FUNCTION_BLOCK "FB_Frequency_Inverter"   // FB6, LAD
{ S7_Optimized_Access := 'TRUE' }
// stored: AutoNumber false, MemoryReserve 100, SetENOAutomatically false
   VAR_INPUT
      Emergency_Stop_Release : Bool;
      Start : Bool;
      Manual_Turn_On_Motor : Bool;
      Pause_Conveyor_Belt_And_Carousel_Functional_Test : Bool;
      Select_Motor_Speedy : SInt;
   END_VAR
   VAR_OUTPUT
      Motor_Spining_Speedy_1 : Bool;
      Motor_Spining_Speedy_2 : Bool;
      Motor_Spining_Speedy_3 : Bool;
   END_VAR
BEGIN

REGION Network 1
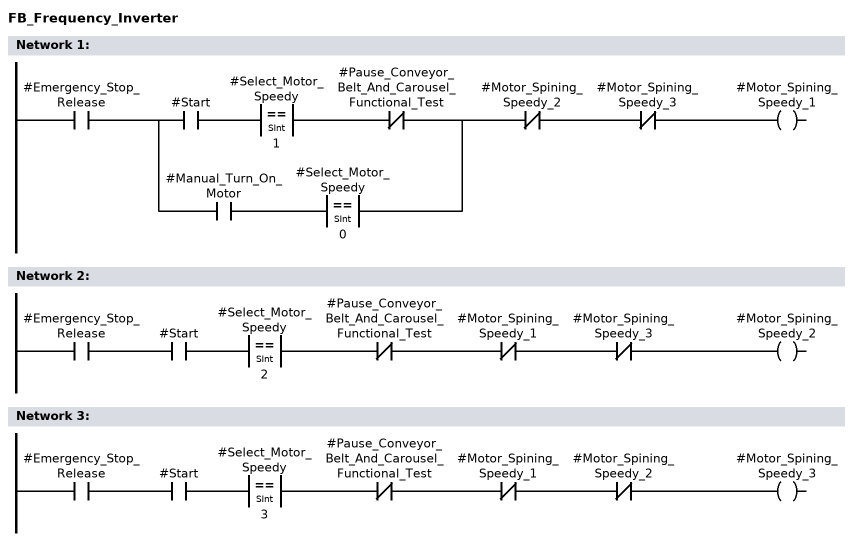
   RUNG wire#powerrail
      Contact( #Emergency_Stop_Release )
      wire#w1
      Contact( #Start )
      { S7_Templates := "SrcType := SInt" } EQ_Contact(in1 := #Select_Motor_Speedy, in2 := 1)
      I_Contact( #Pause_Conveyor_Belt_And_Carousel_Functional_Test )
      wire#w2
      I_Contact( #Motor_Spining_Speedy_2 )
      I_Contact( #Motor_Spining_Speedy_3 )
      Coil( #Motor_Spining_Speedy_1 )
   END_RUNG
   RUNG wire#w1
      Contact( #Manual_Turn_On_Motor )
      { S7_Templates := "SrcType := SInt" } EQ_Contact(in1 := #Select_Motor_Speedy, in2 := 0)
   END_RUNG wire#w2
   // the same network as SCL:
   #Motor_Spining_Speedy_1 := #Emergency_Stop_Release AND ((#Start AND (#Select_Motor_Speedy = 1) AND NOT #Pause_Conveyor_Belt_And_Carousel_Functional_Test) OR (#Manual_Turn_On_Motor AND (#Select_Motor_Speedy = 0))) AND NOT #Motor_Spining_Speedy_2 AND NOT #Motor_Spining_Speedy_3;
END_REGION

REGION Network 2
   RUNG wire#powerrail
      Contact( #Emergency_Stop_Release )
      Contact( #Start )
      { S7_Templates := "SrcType := SInt" } EQ_Contact(in1 := #Select_Motor_Speedy, in2 := 2)
      I_Contact( #Pause_Conveyor_Belt_And_Carousel_Functional_Test )
      I_Contact( #Motor_Spining_Speedy_1 )
      I_Contact( #Motor_Spining_Speedy_3 )
      Coil( #Motor_Spining_Speedy_2 )
   END_RUNG
   // the same network as SCL:
   #Motor_Spining_Speedy_2 := #Emergency_Stop_Release AND #Start AND (#Select_Motor_Speedy = 2) AND NOT #Pause_Conveyor_Belt_And_Carousel_Functional_Test AND NOT #Motor_Spining_Speedy_1 AND NOT #Motor_Spining_Speedy_3;
END_REGION

REGION Network 3
   RUNG wire#powerrail
      Contact( #Emergency_Stop_Release )
      Contact( #Start )
      { S7_Templates := "SrcType := SInt" } EQ_Contact(in1 := #Select_Motor_Speedy, in2 := 3)
      I_Contact( #Pause_Conveyor_Belt_And_Carousel_Functional_Test )
      I_Contact( #Motor_Spining_Speedy_1 )
      I_Contact( #Motor_Spining_Speedy_2 )
      Coil( #Motor_Spining_Speedy_3 )
   END_RUNG
   // the same network as SCL:
   #Motor_Spining_Speedy_3 := #Emergency_Stop_Release AND #Start AND (#Select_Motor_Speedy = 3) AND NOT #Pause_Conveyor_Belt_And_Carousel_Functional_Test AND NOT #Motor_Spining_Speedy_1 AND NOT #Motor_Spining_Speedy_2;
END_REGION
END_FUNCTION_BLOCK

FUNCTION_BLOCK "FB_Send_Water_Fountain_To_Rework"   // FB7, LAD
{ S7_Optimized_Access := 'TRUE' }
// stored: AutoNumber false, MemoryReserve 100, SetENOAutomatically false
   VAR_INPUT
      Emergency_Stop_Release : Bool;
      Start : Bool;
      Water_Fountain_Fail_Test : Bool;
      Trigger_Read_Serial_Number_Exit_Functional_Test : Bool;
      Sensor_Water_Fountain_Exit_Functional_Test_Spinner_Conveyor_Belt : Bool;
      Sensor_Spinner_Exit_Functional_Test_Position_Withdrawn : Bool;
      Sensor_Spinner_Exit_Functional_Test_Position_Advanced : Bool;
      Sensor_Water_Fountain_Exit_Functional_Test_After_Spinner_Conveyor_Belt : Bool;
      Sensor_Water_Fountain_Geting_Entrace_Rework_Conveyor_Belt_Start : Bool;
   END_VAR
   VAR_OUTPUT
      Turn_On_Conveyor_Belt_Motor_Spinner_Get_Exit_Functional_Test : Bool;
      Valve_Advance_Spinner_Get_Exit_Functional_Test : Bool;
      Pause_Conveyor_Belt_And_Carousel_Functional_Test : Bool;
   END_VAR
   VAR
      Aux_Trig_0 : Bool;
      Aux_Trig_1 : Bool;
      Aux_Trig_2 : Bool;
      Aux_Trig_3 : Bool;
      Aux_Trig_4 : Bool;
      Aux_Trig_5 : Bool;
      Aux_Trig_6 : Bool;
      Aux_Trig_7 : Bool;
      Wait_Clean_Spinner : Bool;
      Wait_Get_In_Spinner : Bool;
      "Counter" : USInt;
      Timer_Delay_Turn_On_Motor_Spinner_Conveyor_Belt { S7_SetPoint := 'True'} : TON_TIME;
   END_VAR
   VAR RETAIN
      Counter_Water_Fountain_Exiting_Functional_Test { S7_SetPoint := 'True'} : CTUD_USINT;
   END_VAR
   VAR_TEMP   // added for the SCL form of the ladder/FBD networks
      _w1 : Bool;
      _w2 : Bool;
   END_VAR
BEGIN

REGION Network 1
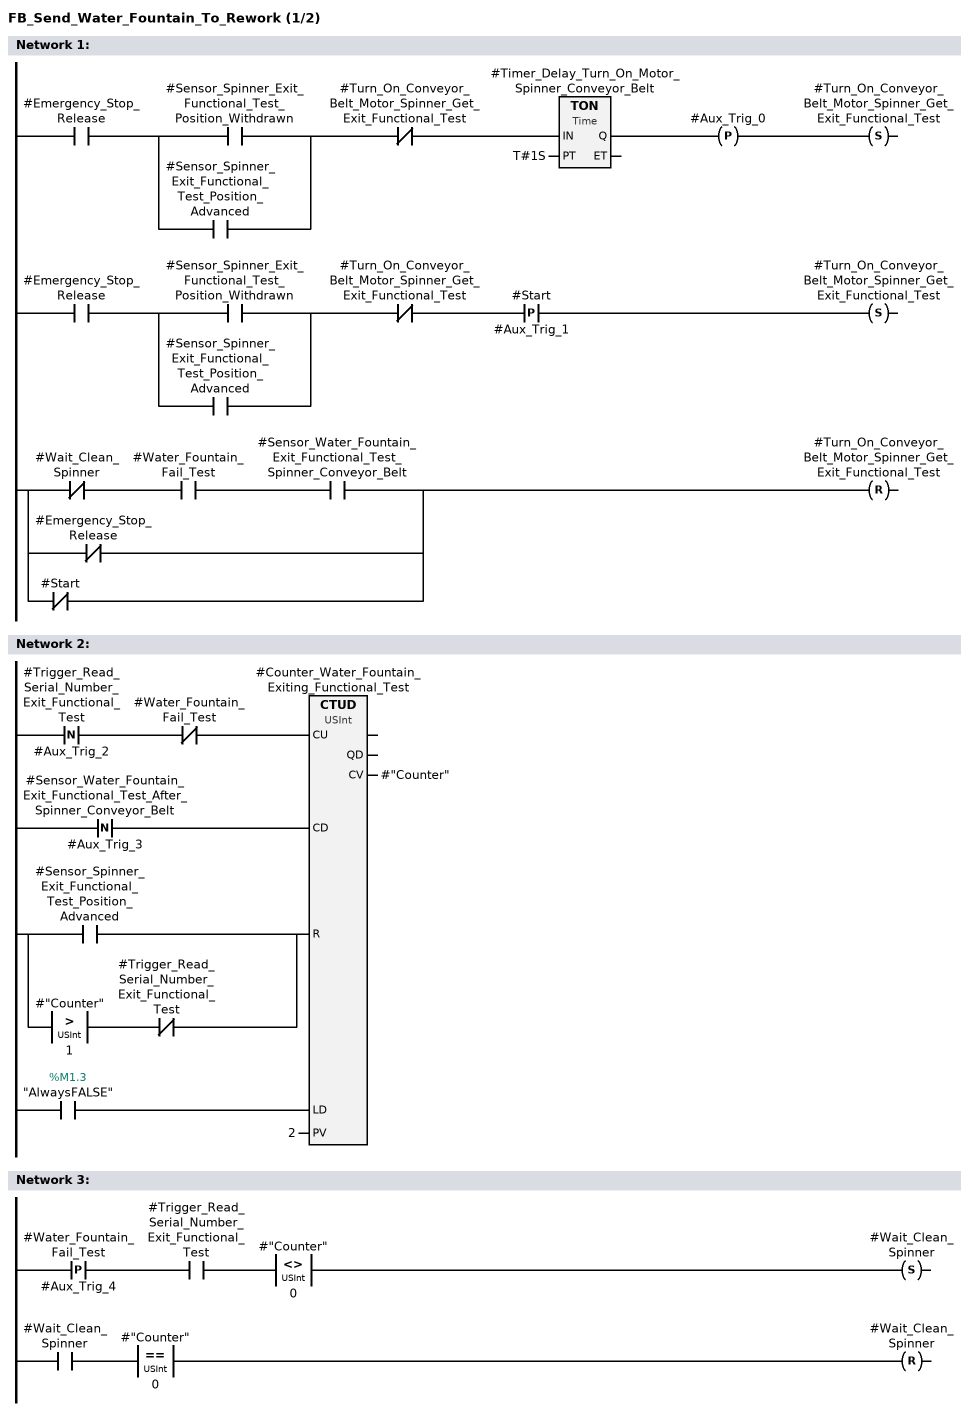
   RUNG wire#powerrail
      Contact( #Emergency_Stop_Release )
      wire#w1
      Contact( #Sensor_Spinner_Exit_Functional_Test_Position_Withdrawn )
      wire#w2
      I_Contact( #Turn_On_Conveyor_Belt_Motor_Spinner_Get_Exit_Functional_Test )
      { S7_Templates := "time_type := Time" } #Timer_Delay_Turn_On_Motor_Spinner_Conveyor_Belt.TON(pt := T#1S, et =>)
      P_Trig( #Aux_Trig_0 )
      S_Coil( #Turn_On_Conveyor_Belt_Motor_Spinner_Get_Exit_Functional_Test )
   END_RUNG
   RUNG wire#w1
      Contact( #Sensor_Spinner_Exit_Functional_Test_Position_Advanced )
   END_RUNG wire#w2
   RUNG wire#powerrail
      Contact( #Emergency_Stop_Release )
      wire#w3
      Contact( #Sensor_Spinner_Exit_Functional_Test_Position_Withdrawn )
      wire#w4
      I_Contact( #Turn_On_Conveyor_Belt_Motor_Spinner_Get_Exit_Functional_Test )
      P_Contact(operand := #Start, bit := #Aux_Trig_1)
      S_Coil( #Turn_On_Conveyor_Belt_Motor_Spinner_Get_Exit_Functional_Test )
   END_RUNG
   RUNG wire#w3
      Contact( #Sensor_Spinner_Exit_Functional_Test_Position_Advanced )
   END_RUNG wire#w4
   RUNG wire#powerrail
      I_Contact( #Wait_Clean_Spinner )
      Contact( #Water_Fountain_Fail_Test )
      Contact( #Sensor_Water_Fountain_Exit_Functional_Test_Spinner_Conveyor_Belt )
      wire#w5
      R_Coil( #Turn_On_Conveyor_Belt_Motor_Spinner_Get_Exit_Functional_Test )
   END_RUNG
   RUNG wire#powerrail
      I_Contact( #Emergency_Stop_Release )
   END_RUNG wire#w5
   RUNG wire#powerrail
      I_Contact( #Start )
   END_RUNG wire#w5
   // the same network as SCL:
   #Timer_Delay_Turn_On_Motor_Spinner_Conveyor_Belt(IN := #Emergency_Stop_Release AND (#Sensor_Spinner_Exit_Functional_Test_Position_Withdrawn OR #Sensor_Spinner_Exit_Functional_Test_Position_Advanced) AND NOT #Turn_On_Conveyor_Belt_Motor_Spinner_Get_Exit_Functional_Test,   // TON
                           PT := T#1S);
   #_w1 := #Timer_Delay_Turn_On_Motor_Spinner_Conveyor_Belt.Q AND NOT #Aux_Trig_0;   // rising edge
   #Aux_Trig_0 := #Timer_Delay_Turn_On_Motor_Spinner_Conveyor_Belt.Q;
   IF #_w1 THEN #Turn_On_Conveyor_Belt_Motor_Spinner_Get_Exit_Functional_Test := TRUE; END_IF;
   #_w2 := #Emergency_Stop_Release AND (#Sensor_Spinner_Exit_Functional_Test_Position_Withdrawn OR #Sensor_Spinner_Exit_Functional_Test_Position_Advanced) AND NOT #Turn_On_Conveyor_Belt_Motor_Spinner_Get_Exit_Functional_Test AND #Start AND NOT #Aux_Trig_1;   // rising edge of #Start
   #Aux_Trig_1 := #Start;
   IF #_w2 THEN #Turn_On_Conveyor_Belt_Motor_Spinner_Get_Exit_Functional_Test := TRUE; END_IF;
   IF (NOT #Wait_Clean_Spinner AND #Water_Fountain_Fail_Test AND #Sensor_Water_Fountain_Exit_Functional_Test_Spinner_Conveyor_Belt) OR NOT #Emergency_Stop_Release OR NOT #Start THEN
       #Turn_On_Conveyor_Belt_Motor_Spinner_Get_Exit_Functional_Test := FALSE;
   END_IF;
END_REGION

REGION Network 2
   RUNG wire#powerrail
      N_Contact(operand := #Trigger_Read_Serial_Number_Exit_Functional_Test, bit := #Aux_Trig_2)
      I_Contact( #Water_Fountain_Fail_Test )
      { S7_Templates := "value_type := USInt" } #Counter_Water_Fountain_Exiting_Functional_Test.CTUD(cd := wire#w1, r := wire#w2, ld := wire#w3, pv := 2, qd =>, cv => #"Counter")
   END_RUNG
   RUNG wire#powerrail
      N_Contact(operand := #Sensor_Water_Fountain_Exit_Functional_Test_After_Spinner_Conveyor_Belt, bit := #Aux_Trig_3)
   END_RUNG wire#w1
   RUNG wire#powerrail
      Contact( #Sensor_Spinner_Exit_Functional_Test_Position_Advanced )
   END_RUNG wire#w2
   RUNG wire#powerrail
      { S7_Templates := "SrcType := USInt" } GT_Contact(in1 := #"Counter", in2 := 1)
      I_Contact( #Trigger_Read_Serial_Number_Exit_Functional_Test )
   END_RUNG wire#w2
   RUNG wire#powerrail
      Contact( "AlwaysFALSE" )
   END_RUNG wire#w3
   // the same network as SCL:
   #_w1 := NOT #Trigger_Read_Serial_Number_Exit_Functional_Test AND #Aux_Trig_2;   // falling edge of #Trigger_Read_Serial_Number_Exit_Functional_Test
   #Aux_Trig_2 := #Trigger_Read_Serial_Number_Exit_Functional_Test;
   #_w2 := NOT #Sensor_Water_Fountain_Exit_Functional_Test_After_Spinner_Conveyor_Belt AND #Aux_Trig_3;   // falling edge of #Sensor_Water_Fountain_Exit_Functional_Test_After_Spinner_Conveyor_Belt
   #Aux_Trig_3 := #Sensor_Water_Fountain_Exit_Functional_Test_After_Spinner_Conveyor_Belt;
   #Counter_Water_Fountain_Exiting_Functional_Test(CU := #_w1 AND NOT #Water_Fountain_Fail_Test,   // CTUD
                           CD := #_w2,
                           R := #Sensor_Spinner_Exit_Functional_Test_Position_Advanced OR ((#"Counter" > 1) AND NOT #Trigger_Read_Serial_Number_Exit_Functional_Test),
                           LD := "AlwaysFALSE",
                           PV := 2,
                           CV => #"Counter");
END_REGION

REGION Network 3
   RUNG wire#powerrail
      P_Contact(operand := #Water_Fountain_Fail_Test, bit := #Aux_Trig_4)
      Contact( #Trigger_Read_Serial_Number_Exit_Functional_Test )
      { S7_Templates := "SrcType := USInt" } NE_Contact(in1 := #"Counter", in2 := 0)
      S_Coil( #Wait_Clean_Spinner )
   END_RUNG
   RUNG wire#powerrail
      Contact( #Wait_Clean_Spinner )
      { S7_Templates := "SrcType := USInt" } EQ_Contact(in1 := #"Counter", in2 := 0)
      R_Coil( #Wait_Clean_Spinner )
   END_RUNG
   // the same network as SCL:
   #_w1 := #Water_Fountain_Fail_Test AND NOT #Aux_Trig_4;   // rising edge of #Water_Fountain_Fail_Test
   #Aux_Trig_4 := #Water_Fountain_Fail_Test;
   IF #_w1 AND #Trigger_Read_Serial_Number_Exit_Functional_Test AND (#"Counter" <> 0) THEN
       #Wait_Clean_Spinner := TRUE;
   END_IF;
   IF #Wait_Clean_Spinner AND (#"Counter" = 0) THEN #Wait_Clean_Spinner := FALSE; END_IF;
END_REGION

REGION Network 4
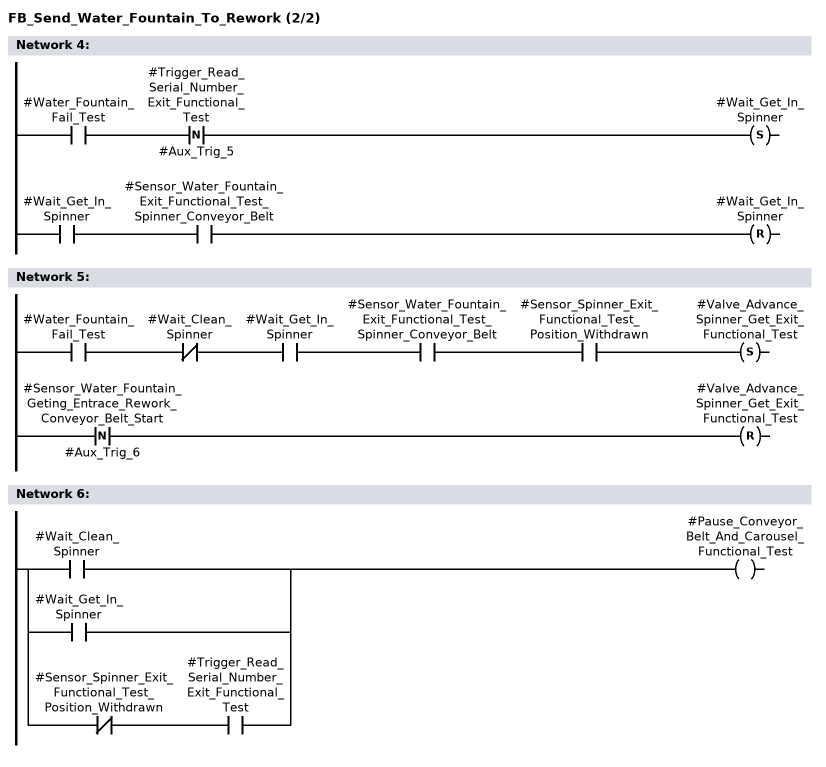
   RUNG wire#powerrail
      Contact( #Water_Fountain_Fail_Test )
      N_Contact(operand := #Trigger_Read_Serial_Number_Exit_Functional_Test, bit := #Aux_Trig_5)
      S_Coil( #Wait_Get_In_Spinner )
   END_RUNG
   RUNG wire#powerrail
      Contact( #Wait_Get_In_Spinner )
      Contact( #Sensor_Water_Fountain_Exit_Functional_Test_Spinner_Conveyor_Belt )
      R_Coil( #Wait_Get_In_Spinner )
   END_RUNG
   // the same network as SCL:
   #_w1 := #Water_Fountain_Fail_Test AND NOT #Trigger_Read_Serial_Number_Exit_Functional_Test AND #Aux_Trig_5;   // falling edge of #Trigger_Read_Serial_Number_Exit_Functional_Test
   #Aux_Trig_5 := #Trigger_Read_Serial_Number_Exit_Functional_Test;
   IF #_w1 THEN #Wait_Get_In_Spinner := TRUE; END_IF;
   IF #Wait_Get_In_Spinner AND #Sensor_Water_Fountain_Exit_Functional_Test_Spinner_Conveyor_Belt THEN
       #Wait_Get_In_Spinner := FALSE;
   END_IF;
END_REGION

REGION Network 5
   RUNG wire#powerrail
      Contact( #Water_Fountain_Fail_Test )
      I_Contact( #Wait_Clean_Spinner )
      Contact( #Wait_Get_In_Spinner )
      Contact( #Sensor_Water_Fountain_Exit_Functional_Test_Spinner_Conveyor_Belt )
      Contact( #Sensor_Spinner_Exit_Functional_Test_Position_Withdrawn )
      S_Coil( #Valve_Advance_Spinner_Get_Exit_Functional_Test )
   END_RUNG
   RUNG wire#powerrail
      N_Contact(operand := #Sensor_Water_Fountain_Geting_Entrace_Rework_Conveyor_Belt_Start, bit := #Aux_Trig_6)
      R_Coil( #Valve_Advance_Spinner_Get_Exit_Functional_Test )
   END_RUNG
   // the same network as SCL:
   IF #Water_Fountain_Fail_Test AND NOT #Wait_Clean_Spinner AND #Wait_Get_In_Spinner AND #Sensor_Water_Fountain_Exit_Functional_Test_Spinner_Conveyor_Belt AND #Sensor_Spinner_Exit_Functional_Test_Position_Withdrawn THEN
       #Valve_Advance_Spinner_Get_Exit_Functional_Test := TRUE;
   END_IF;
   #_w1 := NOT #Sensor_Water_Fountain_Geting_Entrace_Rework_Conveyor_Belt_Start AND #Aux_Trig_6;   // falling edge of #Sensor_Water_Fountain_Geting_Entrace_Rework_Conveyor_Belt_Start
   #Aux_Trig_6 := #Sensor_Water_Fountain_Geting_Entrace_Rework_Conveyor_Belt_Start;
   IF #_w1 THEN #Valve_Advance_Spinner_Get_Exit_Functional_Test := FALSE; END_IF;
END_REGION

REGION Network 6
   RUNG wire#powerrail
      Contact( #Wait_Clean_Spinner )
      wire#w1
      Coil( #Pause_Conveyor_Belt_And_Carousel_Functional_Test )
   END_RUNG
   RUNG wire#powerrail
      Contact( #Wait_Get_In_Spinner )
   END_RUNG wire#w1
   RUNG wire#powerrail
      I_Contact( #Sensor_Spinner_Exit_Functional_Test_Position_Withdrawn )
      Contact( #Trigger_Read_Serial_Number_Exit_Functional_Test )
   END_RUNG wire#w1
   // the same network as SCL:
   #Pause_Conveyor_Belt_And_Carousel_Functional_Test := #Wait_Clean_Spinner OR #Wait_Get_In_Spinner OR (NOT #Sensor_Spinner_Exit_Functional_Test_Position_Withdrawn AND #Trigger_Read_Serial_Number_Exit_Functional_Test);
END_REGION
END_FUNCTION_BLOCK

FUNCTION_BLOCK "FB_Get_Out_Rework_Conveyor_Belt"   // FB8, LAD
{ S7_Optimized_Access := 'TRUE' }
// stored: AutoNumber false, MemoryReserve 100, SetENOAutomatically false
   VAR_INPUT
      Emergency_Stop_Release : Bool;
      Sensor_Water_Fountain_Geting_Exit_Rework_Conveyor_Belt : Bool;
      Button_Water_Fountain_Get_Exit_Rework_Conveyor_Belt : Bool;
      Sensor_Spinner_Entrace_Functional_Test_Position_Advanced : Bool;
      Sensor_Water_Fountain_Entrace_Functional_Test_Spinner_Conveyor_Belt : Bool;
   END_VAR
   VAR_OUTPUT
      Turn_On_Conveyor_Belt_Motor_Rework_Conveyor_Belt_Get_Entrace_Functional_Test : Bool;
   END_VAR
   VAR
      Aux_Trig_0 : Bool;
      Aux_Trig_1 : Bool;
      Aux_Trig_2 : Bool;
      Aux_Trig_3 : Bool;
      Aux_Trig_4 : Bool;
      Aux_Trig_5 : Bool;
      Aux_Trig_6 : Bool;
      Aux_Trig_7 : Bool;
      Button_Is_Pressed : Bool;
   END_VAR
BEGIN

REGION Network 1
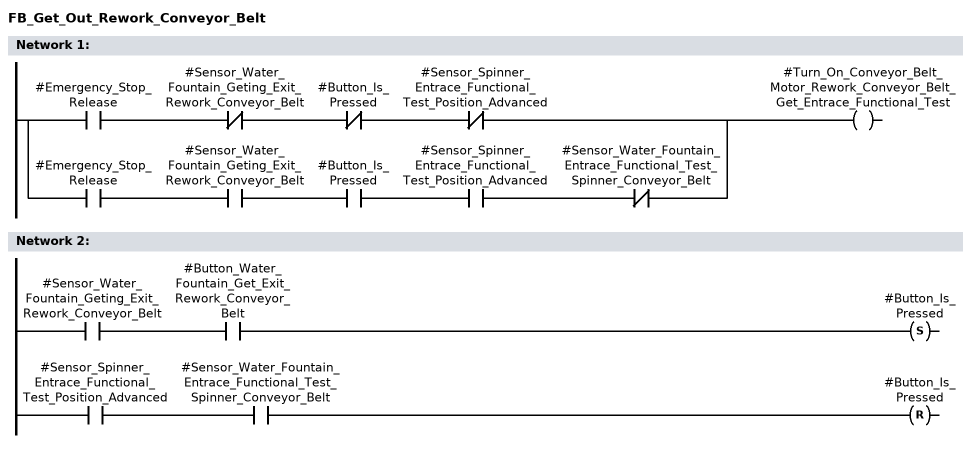
   RUNG wire#powerrail
      Contact( #Emergency_Stop_Release )
      I_Contact( #Sensor_Water_Fountain_Geting_Exit_Rework_Conveyor_Belt )
      I_Contact( #Button_Is_Pressed )
      I_Contact( #Sensor_Spinner_Entrace_Functional_Test_Position_Advanced )
      wire#w1
      Coil( #Turn_On_Conveyor_Belt_Motor_Rework_Conveyor_Belt_Get_Entrace_Functional_Test )
   END_RUNG
   RUNG wire#powerrail
      Contact( #Emergency_Stop_Release )
      Contact( #Sensor_Water_Fountain_Geting_Exit_Rework_Conveyor_Belt )
      Contact( #Button_Is_Pressed )
      Contact( #Sensor_Spinner_Entrace_Functional_Test_Position_Advanced )
      I_Contact( #Sensor_Water_Fountain_Entrace_Functional_Test_Spinner_Conveyor_Belt )
   END_RUNG wire#w1
   // the same network as SCL:
   #Turn_On_Conveyor_Belt_Motor_Rework_Conveyor_Belt_Get_Entrace_Functional_Test := (#Emergency_Stop_Release AND NOT #Sensor_Water_Fountain_Geting_Exit_Rework_Conveyor_Belt AND NOT #Button_Is_Pressed AND NOT #Sensor_Spinner_Entrace_Functional_Test_Position_Advanced) OR (#Emergency_Stop_Release AND #Sensor_Water_Fountain_Geting_Exit_Rework_Conveyor_Belt AND #Button_Is_Pressed AND #Sensor_Spinner_Entrace_Functional_Test_Position_Advanced AND NOT #Sensor_Water_Fountain_Entrace_Functional_Test_Spinner_Conveyor_Belt);
END_REGION

REGION Network 2
   RUNG wire#powerrail
      Contact( #Sensor_Water_Fountain_Geting_Exit_Rework_Conveyor_Belt )
      Contact( #Button_Water_Fountain_Get_Exit_Rework_Conveyor_Belt )
      S_Coil( #Button_Is_Pressed )
   END_RUNG
   RUNG wire#powerrail
      Contact( #Sensor_Spinner_Entrace_Functional_Test_Position_Advanced )
      Contact( #Sensor_Water_Fountain_Entrace_Functional_Test_Spinner_Conveyor_Belt )
      R_Coil( #Button_Is_Pressed )
   END_RUNG
   // the same network as SCL:
   IF #Sensor_Water_Fountain_Geting_Exit_Rework_Conveyor_Belt AND #Button_Water_Fountain_Get_Exit_Rework_Conveyor_Belt THEN
       #Button_Is_Pressed := TRUE;
   END_IF;
   IF #Sensor_Spinner_Entrace_Functional_Test_Position_Advanced AND #Sensor_Water_Fountain_Entrace_Functional_Test_Spinner_Conveyor_Belt THEN
       #Button_Is_Pressed := FALSE;
   END_IF;
END_REGION
END_FUNCTION_BLOCK

FUNCTION_BLOCK "FB_Get_In_Rework_Conveyor_Belt"   // FB9, LAD
{ S7_Optimized_Access := 'TRUE' }
// stored: AutoNumber false, MemoryReserve 100, SetENOAutomatically false
   VAR_INPUT
      Emergency_Stop_Release : Bool;
      Start : Bool;
      Sensor_Water_Fountain_Exit_Functional_Test_Spinner_Conveyor_Belt : Bool;
      Sensor_Spinner_Exit_Functional_Test_Position_Withdrawn : Bool;
      Sensor_Spinner_Exit_Functional_Test_Position_Advanced : Bool;
      Sensor_Water_Fountain_Geting_Entrace_Rework_Conveyor_Belt_Start : Bool;
      Sensor_Water_Fountain_Geting_Entrace_Rework_Conveyor_Belt_Finish : Bool;
   END_VAR
   VAR_OUTPUT
      Turn_On_Conveyor_Belt_Motor_Rework_Conveyor_Belt_Get_Exit_Funcional_Test : Bool;
   END_VAR
BEGIN

REGION Network 1
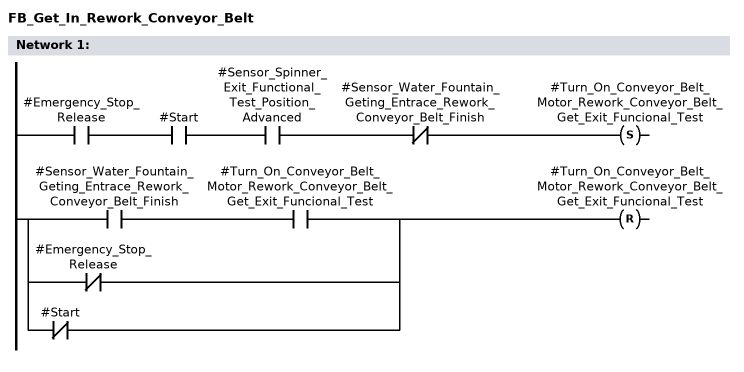
   RUNG wire#powerrail
      Contact( #Emergency_Stop_Release )
      Contact( #Start )
      Contact( #Sensor_Spinner_Exit_Functional_Test_Position_Advanced )
      I_Contact( #Sensor_Water_Fountain_Geting_Entrace_Rework_Conveyor_Belt_Finish )
      S_Coil( #Turn_On_Conveyor_Belt_Motor_Rework_Conveyor_Belt_Get_Exit_Funcional_Test )
   END_RUNG
   RUNG wire#powerrail
      Contact( #Sensor_Water_Fountain_Geting_Entrace_Rework_Conveyor_Belt_Finish )
      Contact( #Turn_On_Conveyor_Belt_Motor_Rework_Conveyor_Belt_Get_Exit_Funcional_Test )
      wire#w1
      R_Coil( #Turn_On_Conveyor_Belt_Motor_Rework_Conveyor_Belt_Get_Exit_Funcional_Test )
   END_RUNG
   RUNG wire#powerrail
      I_Contact( #Emergency_Stop_Release )
   END_RUNG wire#w1
   RUNG wire#powerrail
      I_Contact( #Start )
   END_RUNG wire#w1
   // the same network as SCL:
   IF #Emergency_Stop_Release AND #Start AND #Sensor_Spinner_Exit_Functional_Test_Position_Advanced AND NOT #Sensor_Water_Fountain_Geting_Entrace_Rework_Conveyor_Belt_Finish THEN
       #Turn_On_Conveyor_Belt_Motor_Rework_Conveyor_Belt_Get_Exit_Funcional_Test := TRUE;
   END_IF;
   IF (#Sensor_Water_Fountain_Geting_Entrace_Rework_Conveyor_Belt_Finish AND #Turn_On_Conveyor_Belt_Motor_Rework_Conveyor_Belt_Get_Exit_Funcional_Test) OR NOT #Emergency_Stop_Release OR NOT #Start THEN
       #Turn_On_Conveyor_Belt_Motor_Rework_Conveyor_Belt_Get_Exit_Funcional_Test := FALSE;
   END_IF;
END_REGION
END_FUNCTION_BLOCK

FUNCTION_BLOCK "FB_Caroussel_Voltage_Selection"   // FB10, LAD
{ S7_Optimized_Access := 'TRUE' }
// stored: MemoryReserve 100, SetENOAutomatically false
   VAR_INPUT
      Emergency_Stop_Release : Bool;
      Selected_Voltage_220V : Bool;
      Selected_Voltage_127V : Bool;
      Carousel_Voltage_Selection : SInt;
   END_VAR
   VAR_OUTPUT
      Voltage_220V_Selected : Bool;
      Voltage_127V_Selected : Bool;
   END_VAR
   VAR
      Delay_Turn_On_220V { S7_SetPoint := 'True'} : TON_TIME;
      Delay_Turn_On_127V { S7_SetPoint := 'True'} : TON_TIME;
   END_VAR
BEGIN

REGION Network 1
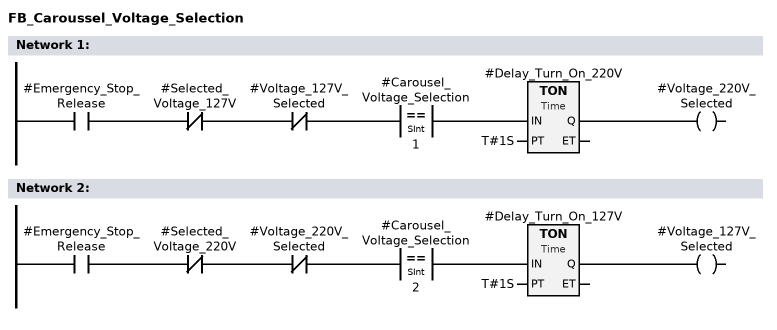
   RUNG wire#powerrail
      Contact( #Emergency_Stop_Release )
      I_Contact( #Selected_Voltage_127V )
      I_Contact( #Voltage_127V_Selected )
      { S7_Templates := "SrcType := SInt" } EQ_Contact(in1 := #Carousel_Voltage_Selection, in2 := 1)
      { S7_Templates := "time_type := Time" } #Delay_Turn_On_220V.TON(pt := T#1S, et =>)
      Coil( #Voltage_220V_Selected )
   END_RUNG
   // the same network as SCL:
   #Delay_Turn_On_220V(IN := #Emergency_Stop_Release AND NOT #Selected_Voltage_127V AND NOT #Voltage_127V_Selected AND (#Carousel_Voltage_Selection = 1),   // TON
                       PT := T#1S);
   #Voltage_220V_Selected := #Delay_Turn_On_220V.Q;
END_REGION

REGION Network 2
   RUNG wire#powerrail
      Contact( #Emergency_Stop_Release )
      I_Contact( #Selected_Voltage_220V )
      I_Contact( #Voltage_220V_Selected )
      { S7_Templates := "SrcType := SInt" } EQ_Contact(in1 := #Carousel_Voltage_Selection, in2 := 2)
      { S7_Templates := "time_type := Time" } #Delay_Turn_On_127V.TON(pt := T#1S, et =>)
      Coil( #Voltage_127V_Selected )
   END_RUNG
   // the same network as SCL:
   #Delay_Turn_On_127V(IN := #Emergency_Stop_Release AND NOT #Selected_Voltage_220V AND NOT #Voltage_220V_Selected AND (#Carousel_Voltage_Selection = 2),   // TON
                       PT := T#1S);
   #Voltage_127V_Selected := #Delay_Turn_On_127V.Q;
END_REGION
END_FUNCTION_BLOCK

DATA_BLOCK "Instance_FB_Caroussel_Voltage_Selection_DB"   // DB111
// stored: AutoNumber false, InstanceOfName FB_Caroussel_Voltage_Selection, InstanceOfType FB
"FB_Caroussel_Voltage_Selection"
BEGIN
END_DATA_BLOCK

DATA_BLOCK "Instance_FB_Digital_Input_DB"   // DB101
// stored: AutoNumber false, InstanceOfName FB_Digital_Input, InstanceOfType FB
"FB_Digital_Input"
BEGIN
END_DATA_BLOCK

DATA_BLOCK "Instance_FB_Digital_Output_DB"   // DB103
// stored: AutoNumber false, InstanceOfName FB_Digital_Output, InstanceOfType FB
"FB_Digital_Output"
BEGIN
END_DATA_BLOCK

DATA_BLOCK "Instance_FB_Frequency_Inverter_DB_Conveyor_Belt"   // DB107
// stored: AutoNumber false, InstanceOfName FB_Frequency_Inverter, InstanceOfType FB
"FB_Frequency_Inverter"
BEGIN
END_DATA_BLOCK

DATA_BLOCK "Instance_FB_Frequency_Inverter_DB_Spin_Caroussel"   // DB106
// stored: AutoNumber false, InstanceOfName FB_Frequency_Inverter, InstanceOfType FB
"FB_Frequency_Inverter"
BEGIN
END_DATA_BLOCK

DATA_BLOCK "Instance_FB_Get_In_Rework_Conveyor_Belt_DB"   // DB110
// stored: AutoNumber false, InstanceOfName FB_Get_In_Rework_Conveyor_Belt, InstanceOfType FB
"FB_Get_In_Rework_Conveyor_Belt"
BEGIN
END_DATA_BLOCK

DATA_BLOCK "Instance_FB_Get_Out_Rework_Conveyor_Belt_DB"   // DB109
// stored: AutoNumber false, InstanceOfName FB_Get_Out_Rework_Conveyor_Belt, InstanceOfType FB
"FB_Get_Out_Rework_Conveyor_Belt"
BEGIN
END_DATA_BLOCK

DATA_BLOCK "Instance_FB_IO_Device_DB"   // DB104
// stored: AutoNumber false, InstanceOfName FB_IO_Device, InstanceOfType FB
"FB_IO_Device"
BEGIN
END_DATA_BLOCK

DATA_BLOCK "Instance_FB_Recive_Water_Fountain_From_Rework_DB"   // DB105
// stored: AutoNumber false, InstanceOfName FB_Recive_Water_Fountain_From_Rework, InstanceOfType FB
"FB_Recive_Water_Fountain_From_Rework"
BEGIN
END_DATA_BLOCK

DATA_BLOCK "Instance_FB_Send_Water_Fountain_To_Rework_DB"   // DB108
// stored: AutoNumber false, InstanceOfName FB_Send_Water_Fountain_To_Rework, InstanceOfType FB
"FB_Send_Water_Fountain_To_Rework"
BEGIN
END_DATA_BLOCK
